(* IEC 61131-3 sources: JaccoSigma/tempclass/Class/Send_Message, 1 file *)

(* ---- Send_Message.st ---- *)
#pragma usingLtd DSComm_Interface

(*!
<Class
	Name               = "Send_Message"
	Revision           = "0.0"
	RealtimeTask       = "false"
	CyclicTask         = "false"
	BackgroundTask     = "true"
	DefBackground      = "1000 ms"
	Sigmatek           = "false"
	OSInterface        = "false"
	HighPriority       = "false"
	Automatic          = "false"
	UpdateMode         = "Prescan"
	SharedCommandTable = "true"
	Objectsize         = "(340,120)">
	<Channels>
		<Server Name="ClassSvr" Visualized="false" Initialize="false" WriteProtected="false" Retentive="false"/>
		<Client Name="DSComm" Required="true" Internal="false"/>
		<Client Name="Link_E" Required="true" Internal="false"/>
		<Client Name="SigCLib" Required="false" Internal="false"/>
	</Channels>
</Class>
*)
Send_Message : CLASS
  //Servers:
	ClassSvr 	: SvrChCmd_DINT;
  //Clients:
	Link_E 	: CltChCmd_DSComm_Eventjournal;
	SigCLib 	: CltChCmd_SigCLib;
	DSComm 	: CltChCmd_DSComm;
  //Variables:
		retcode 	: DINT;
		Variable 	: DINT;
  //Functions:

	FUNCTION VIRTUAL GLOBAL Background
		VAR_INPUT
			EAX 	: UDINT;
		END_VAR
		VAR_OUTPUT
			state (EAX) 	: UDINT;
		END_VAR;

	FUNCTION VIRTUAL GLOBAL ClassSvr::Write
		VAR_INPUT
			input (EAX) 	: DINT;
		END_VAR
		VAR_OUTPUT
			result (EAX) 	: DINT;
		END_VAR;
  //Tables:
	FUNCTION @STD
		VAR_OUTPUT
			ret_code	: CONFSTATES;
		END_VAR;
	FUNCTION GLOBAL TAB @CT_;
END_CLASS;

#pragma usingLtd DSComm
#pragma usingLtd DSComm_Eventjournal
#pragma usingLtd SigCLib

//werkt niet

FUNCTION VIRTUAL GLOBAL Send_Message::ClassSvr::Write
	VAR_INPUT
		input (EAX) 	: DINT;
	END_VAR
	VAR_OUTPUT
		result (EAX) 	: DINT;
	END_VAR
  VAR
  	pText : ^CHAR;
  END_VAR

  ClassSvr := input;

  pText := "12345";
  ClassSvr := Link_E.AddMessage(pText:=pText$^UINT, textLength:=5, charSize:=sizeof(_ASCII));

	result := ClassSvr;

END_FUNCTION

FUNCTION VIRTUAL GLOBAL Send_Message::Background
	VAR_INPUT
		EAX 	: UDINT;
	END_VAR
	VAR_OUTPUT
		state (EAX) 	: UDINT;
	END_VAR
    VAR
    username : array [0..15] of uint;
    password : array [0..15] of uint;
  END_VAR

  if Variable = 0 then
    sigclib_tostr16(dst0:=#username[0], src0:="superuser");
    sigclib_tostr16(dst0:=#password[0], src0:="sigmatek");

    retcode := DSComm.UserLogin(pThis:=Link_E.pCh$^DSComm_Interface, pUserName:=#username[0], pPassword:=#password[0]);
    Variable := 1;
  end_if;

	state := READY;

END_FUNCTION
